FUNCTION_BLOCK Led
VAR
	_state : BOOL;
END_VAR

PROPERTY State : BOOL
GET
State := _state;
END_GET
SET
_state := State;
END_SET
END_PROPERTY

END_FUNCTION_BLOCK

(* stored: Version 1.1.0.1, ProductVersion 3.1.4024.12
   POU Led: Id {eee83838-3c2c-43ec-8b89-683878a85abd}, SpecialFunc None
   Property State: Id {e3a1b6cd-cb48-465d-b773-1a08ffdb9242}
   Get Get: Id {36c5ca79-529f-4892-bf03-3de869524f7e}
   Set Set: Id {4324096c-7237-4c8f-8743-ad9168051b93} *)
